FUNCTION FUN_ITR : LREAL
VAR_INPUT
	N: INT;
END_VAR
VAR
END_VAR

FUN_ITR:= (INT_TO_LREAL(N)/32767)*200000;

END_FUNCTION

(* stored: Version 1.1.0.1, ProductVersion 3.1.4022.16
   POU FUN_ITR: Id {f309a4ca-9f43-4ec4-892b-39abe8429e43}, SpecialFunc None *)
